(* CoDeSys 2.3.9.50 project: Luftkanal.pro *)
(* Libraries: STANDARD.LIB 5.6.98 12:03:02 *)

(* Task configuration *)
TASK Standard (PRIORITY := 0, INTERVAL := T#10ms);
	MAIN
END_TASK

(* POU MAIN, ST *)
PROGRAM MAIN
VAR


	b_butYellow		AT %I*	:BOOL;			(* Yellow button *)
	b_butBlue		AT %I*	:BOOL;			(* Blue button *)
	b_lampRed		AT %Q*	:BOOL:=TRUE;	(* Red lamp *)
	b_lampGreen		AT %Q*	:BOOL;			(* Green lamp *)
	i_anDisp		AT %Q*	:INT;			(* Analog meter *)

	ui_heatControl	AT %Q*	:USINT;
	i_heatDuty		AT %Q*	:INT;
	ui_fanControl	AT %Q*	:USINT;
	i_fanDuty		AT %Q*	:INT;

	i_temp			AT %I*	:INT;

END_VAR
IF b_butYellow = TRUE THEN			(* Turn on with yellow button *)
	b_lampGreen := TRUE;
	b_lampRed := FALSE;


END_IF

IF b_butBLUE = TRUE THEN			(* Turn off*)
	b_lampRed := TRUE;
	b_lampGreen := FALSE;
END_IF
END_PROGRAM
